// TIA Portal V18 export
// export: Created 2026-03-12T16:04:35.3493985Z, ExportSetting WithDefaults, DisplayName Totally Integrated Automation Portal, DisplayVersion V18 Update 5, DisplayName TIA Portal Openness, DisplayVersion V18 Update 5, DisplayName TIA Portal Version Control Interface, DisplayVersion V18, DisplayName SINAMICS Startdrive Advanced, DisplayVersion V18, DisplayName SINAMICS Startdrive G130, G150, S120, S150, SINAMICS MV, S210, DisplayVersion V18, DisplayName SINAMICS Startdrive G110M, G120, G120C, G120D, G120P, G115D, DisplayVersion V18, DisplayName STEP 7 Professional, DisplayVersion V18 Update 5, DisplayName STEP 7 Safety, DisplayVersion V18, DisplayName WinCC Professional, DisplayVersion V18 Update 5
FUNCTION_BLOCK "FB SETPOINT ESCALONAMENTO"   // FB13, LAD
TITLE = Function Block SETPOINT L/H TO RPM - Bloco para escalonar o setpoint de uma unidade para rpm
{ S7_Optimized_Access := 'TRUE' }
VERSION : 0.1
// Network 1: Escalonamento dos ranges
// stored: AutoNumber true, IsIECCheckEnabled false, IsRetainMemResEnabled false, MemoryReserve 100, SetENOAutomatically false, UDAEnableTagReadback false
   VAR_INPUT
      MAX_UNIT : Int;   // Unidade máxima para escalonamento
      MAX_RPM_TOTAL : Int;   // RPM total do equipamento
      MAX_RPM_IHM : Int;   // RPM máximo cadastrado pela IHM
      MIN_RPM_IHM : Int;   // RPM mínimo cadastrado pela IHM
   END_VAR
   VAR_OUTPUT
      SETPOINT_UNIT_OUT : Int;   // Setpoint da unidade convertida em rpm
      SETPOINT_UNIT_IN : Int;
   END_VAR
   VAR_IN_OUT
      SETPOINT : Int;   // Setpoint em unidade recebido da IHM
   END_VAR
   VAR RETAIN
      SETPOINT_MIN_UNIT : Int;   // Setpoint mínimo calculado de rpm para unidade
      SETPOINT_MAX_UNIT : Int;   // Setpoint máximo calculado de rpm para unidade
   END_VAR
BEGIN

REGION Network 1: Escalonamento dos ranges
   // MAX_RPM = RPM máximo cadastrado pela IHM
   // MIN_RPM = RPM mínimo cadastrado pela IHM
   // MAX_RPM_TOTAL = Limite físico máximo em rpm dos sopradores
   // MAX_UNIT = Pressão máxima dos sopradores
   // SETPOINT_RPM = Setpoint de milibar convertido em rpm
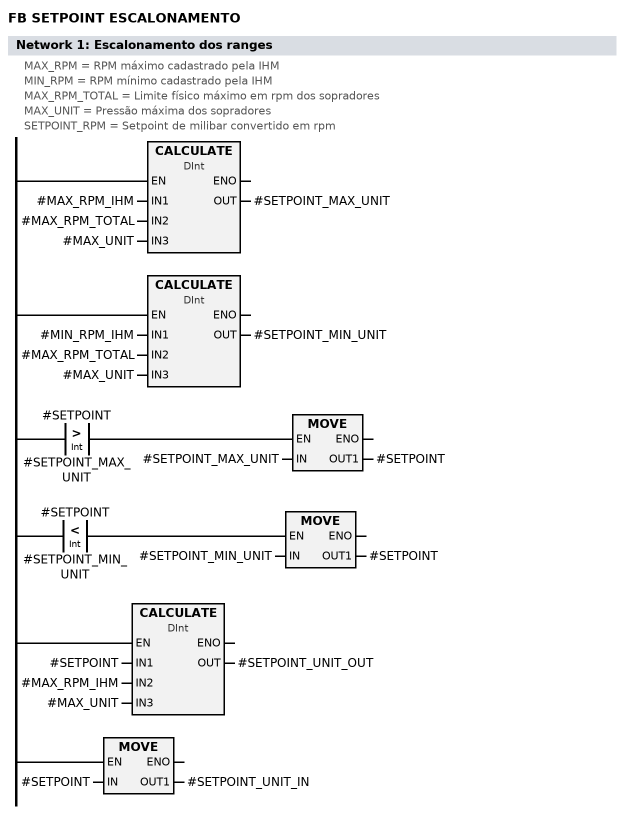
   RUNG wire#powerrail
      { S7_Templates := "SrcType := DInt"; S7_Expression := "(IN1*IN3) / IN2" } Calculate(in1 := #MAX_RPM_IHM, in2 := #MAX_RPM_TOTAL, in3 := #MAX_UNIT, out => #SETPOINT_MAX_UNIT)
   END_RUNG
   RUNG wire#powerrail
      { S7_Templates := "SrcType := DInt"; S7_Expression := "(IN1*IN3) / IN2" } Calculate(in1 := #MIN_RPM_IHM, in2 := #MAX_RPM_TOTAL, in3 := #MAX_UNIT, out => #SETPOINT_MIN_UNIT)
   END_RUNG
   RUNG wire#powerrail
      { S7_Templates := "SrcType := Int" } GT_Contact(in1 := #SETPOINT, in2 := #SETPOINT_MAX_UNIT)
      Move(in := #SETPOINT_MAX_UNIT, out1 => #SETPOINT)
   END_RUNG
   RUNG wire#powerrail
      { S7_Templates := "SrcType := Int" } LT_Contact(in1 := #SETPOINT, in2 := #SETPOINT_MIN_UNIT)
      Move(in := #SETPOINT_MIN_UNIT, out1 => #SETPOINT)
   END_RUNG
   RUNG wire#powerrail
      { S7_Templates := "SrcType := DInt"; S7_Expression := "(IN1*IN2) / IN3" } Calculate(in1 := #SETPOINT, in2 := #MAX_RPM_IHM, in3 := #MAX_UNIT, out => #SETPOINT_UNIT_OUT)
   END_RUNG
   RUNG wire#powerrail
      Move(in := #SETPOINT, out1 => #SETPOINT_UNIT_IN)
   END_RUNG
   // the same network as SCL:
   #SETPOINT_MAX_UNIT := (#MAX_RPM_IHM*#MAX_UNIT) / #MAX_RPM_TOTAL;
   #SETPOINT_MIN_UNIT := (#MIN_RPM_IHM*#MAX_UNIT) / #MAX_RPM_TOTAL;
   IF #SETPOINT > #SETPOINT_MAX_UNIT THEN #SETPOINT := #SETPOINT_MAX_UNIT; END_IF;
   IF #SETPOINT < #SETPOINT_MIN_UNIT THEN #SETPOINT := #SETPOINT_MIN_UNIT; END_IF;
   #SETPOINT_UNIT_OUT := (#SETPOINT*#MAX_RPM_IHM) / #MAX_UNIT;
   #SETPOINT_UNIT_IN := #SETPOINT;
END_REGION
END_FUNCTION_BLOCK
